/// Test case template
FUNCTION_BLOCK INTERNAL FB_TestCaseBase IMPLEMENTS ITestCase
VAR
	/// state of test case
	eState	: E_TestCaseState;
	/// result of test case
	eResult	: E_TestResult;
END_VAR

{attribute 'object_name' := 'Reset'}
METHOD Reset
// reset var's
eState := E_TestCaseState.eTestCaseState_ready;
eResult := E_TestResult.eTestResult_none;
END_METHOD

{attribute 'object_name' := 'Run'}
METHOD Run : E_TestCaseState
// set state to running, if ready
IF eState = E_TestCaseState.eTestCaseState_ready AND eResult = E_TestResult.eTestResult_none THEN
	eState := E_TestCaseState.eTestCaseState_running;
ELSIF eState <> E_TestCaseState.eTestCaseState_running THEN
	eState := E_TestCaseState.eTestCaseState_error;
END_IF

Run := eState;
END_METHOD

{attribute 'monitoring' := 'call'}
PROPERTY TestResult : E_TestResult
GET
TestResult := eResult;
END_GET
END_PROPERTY

{attribute 'monitoring' := 'call'}
PROPERTY TestState : E_TestCaseState
GET
TestState := eState;
END_GET
END_PROPERTY

END_FUNCTION_BLOCK

(* stored: Version 1.1.0.1, ProductVersion 3.1.4024.12
   POU FB_TestCaseBase: Id {1f0dc0dd-a567-4aa1-bc21-370db998da9a}, SpecialFunc None
   Method Reset: Id {0f19a61a-bedf-491c-b539-0a6ac82f1352}
   Method Run: Id {682cf9bd-e5a2-4777-80df-63d898df2a3b}
   Property TestResult: Id {c6c5e47f-9860-4e04-a93c-16c7a3541708}
   Get Get: Id {d1afe8a9-8fce-456f-ab88-74981c29cc4e}
   Property TestState: Id {ed4b6957-bc0d-495d-abd2-ce81fe66878b}
   Get Get: Id {9f2518cc-1b0e-40b4-8a30-981d71d4ed42} *)
